FUNCTION VecNormalize : Vec3
VAR_INPUT
	a : Vec3;
END_VAR
VAR
END_VAR

VecNormalize := VecMulNum(a, 1/VecNorm(a));

END_FUNCTION

(* stored: Version 1.1.0.1, ProductVersion 3.1.4024.2
   POU VecNormalize: Id {7cb7a3c3-0f84-4b9e-8aba-6af6635ab7dc}, SpecialFunc None *)
